PROGRAM Control_FBD
VAR
END_VAR

END_PROGRAM

(* stored: Version 1.1.0.1, ProductVersion 3.1.4022.12
   POU Control_FBD: Id {6577cfd4-7983-4a0a-ac09-462777cb4efb}, SpecialFunc None *)
